// SIMATIC S7-200 project (STEP 7-Micro/WIN), CPU 224 UN REL 02.01

ORGANIZATION_BLOCK 主程序:OB1
TITLE=程序注释
BEGIN
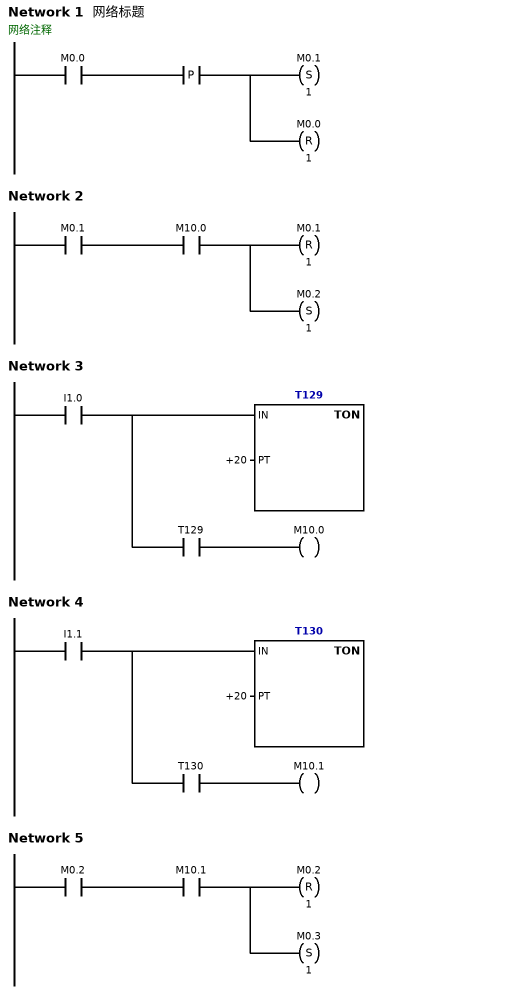
Network 1 // 网络标题
// 网络注释
LD     M0.0
EU
S      M0.1, 1
R      M0.0, 1
Network 2
LD     M0.1
A      M10.0
R      M0.1, 1
S      M0.2, 1
Network 3
LD     I1.0
TON    T129, +20
A      T129
=      M10.0
Network 4
LD     I1.1
TON    T130, +20
A      T130
=      M10.1
Network 5
LD     M0.2
A      M10.1
R      M0.2, 1
S      M0.3, 1
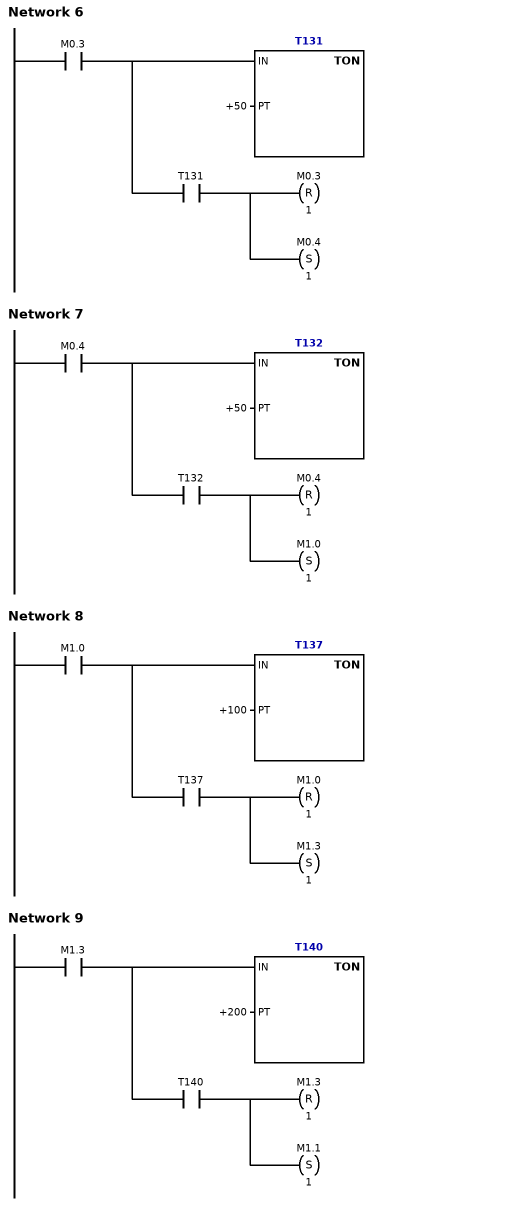
Network 6
LD     M0.3
TON    T131, +50
A      T131
R      M0.3, 1
S      M0.4, 1
Network 7
LD     M0.4
TON    T132, +50
A      T132
R      M0.4, 1
S      M1.0, 1
Network 8
LD     M1.0
TON    T137, +100
A      T137
R      M1.0, 1
S      M1.3, 1
Network 9
LD     M1.3
TON    T140, +200
A      T140
R      M1.3, 1
S      M1.1, 1
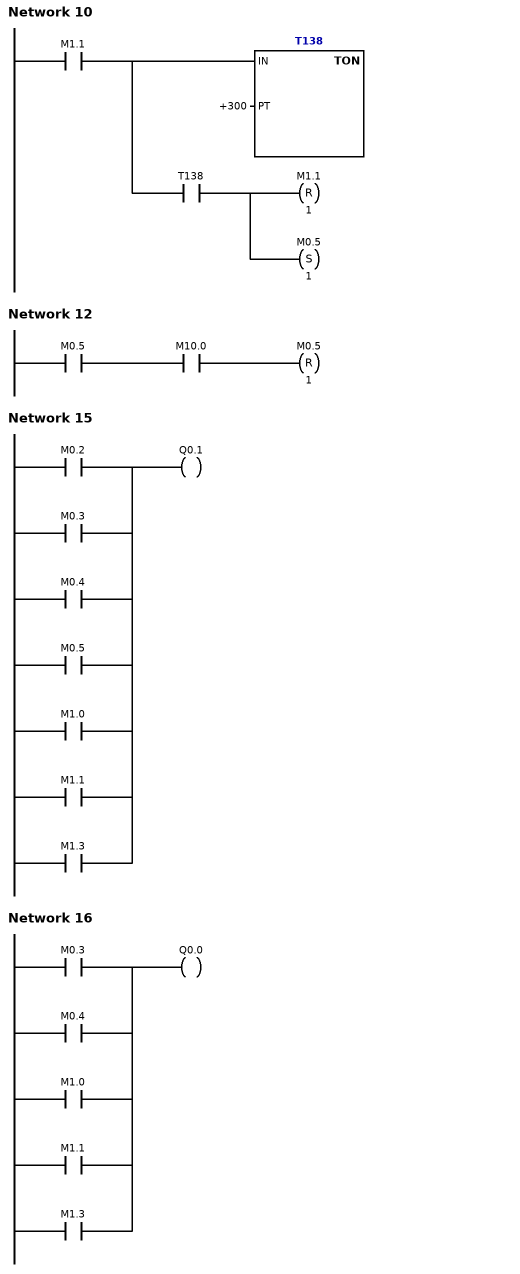
Network 10
LD     M1.1
TON    T138, +300
A      T138
R      M1.1, 1
S      M0.5, 1
Network 12
LD     M0.5
A      M10.0
R      M0.5, 1
Network 15
LD     M0.2
O      M0.3
O      M0.4
O      M0.5
O      M1.0
O      M1.1
O      M1.3
=      Q0.1
Network 16
LD     M0.3
O      M0.4
O      M1.0
O      M1.1
O      M1.3
=      Q0.0
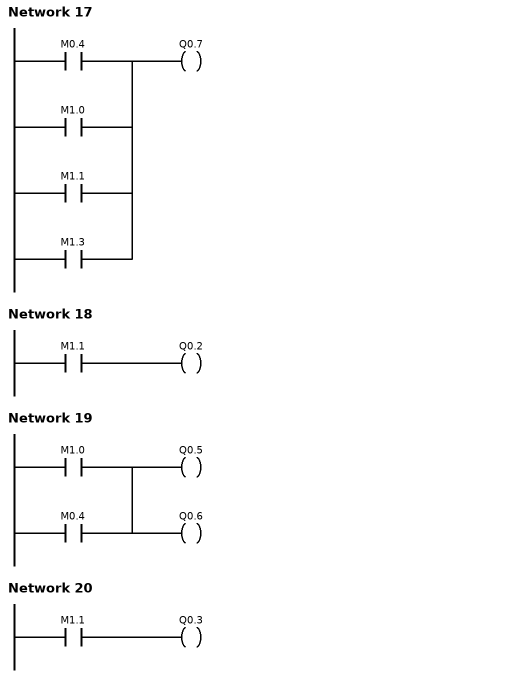
Network 17
LD     M0.4
O      M1.0
O      M1.1
O      M1.3
=      Q0.7
Network 18
LD     M1.1
=      Q0.2
Network 19
LD     M1.0
O      M0.4
=      Q0.5
=      Q0.6
Network 20
LD     M1.1
=      Q0.3
END_ORGANIZATION_BLOCK
